// TIA Portal V21 export
VAR_GLOBAL   // PLC tag table "PallettizzatoreReciveDigitali"
END_VAR
VAR_GLOBAL CONSTANT   // user constants
   K_SegnaleDaPallettizzatore_Marcia : Int := 1;
   K_SegnaleDaPallettizzatore_Pronto : Int := 2;
END_VAR
